PROGRAM P_Modbus
VAR
END_VAR

P_Modbus_RTU();
PRG_SerialComm();

END_PROGRAM

(* stored: Version 1.1.0.1, ProductVersion 3.1.4024.11
   POU P_Modbus: Id {209a01be-f792-42d6-afed-d2e76d07080f}, SpecialFunc None *)
